# EPICS StreamDevice protocol: agilent/hp53181a/device_config/hp53181a.proto
Terminator = CR LF;
ReadTimeout = 500;
ExtraInput = Ignore;

raw_num{
    in "%[0-9,.]";
}

read_unit{
    in "%*[0-9,.]\_%{Hz|MHz}";
}
